(* CoDeSys 2.3 export: ENGINE_TRIPPED.EXP *)

(* POU ENGINE_TRIPPED, ST *)
FUNCTION_BLOCK ENGINE_TRIPPED
VAR_INPUT
END_VAR
VAR_OUTPUT
END_VAR
VAR
END_VAR
IF 	SHUTDOWN = TRUE
	AND	ENG_STANDSTILL_P = TRUE
THEN
	ENGINE_TRIPPED_P := TRUE;
ELSE
	ENGINE_TRIPPED_P := FALSE;
END_IF
END_FUNCTION_BLOCK
